(* IEC 61131-3 sources: TcView/src/tests/regression/golden/fragments, 2 files *)

(* ---- FB_IntegrationSample.Method_FB_Init.st ---- *)
METHOD FB_Init : BOOL
VAR_INPUT
    bInitRetains : BOOL;
END_VAR
// comment in declaration

FB_Init := TRUE;

(* ---- I_IntegrationSample.Method_Reset.st ---- *)
METHOD Reset : BOOL
VAR_INPUT
    bHard : BOOL;
END_VAR
